(* Logix 5000 project; controller LeakTestAuto vendor 1 type 14 code 226 rev 37.11; software revision 37.01; part 14 of 14 *)
(* tags used below, declared in another part *)
   OP220 : udt_Mode;
   OP220_EStop_OK : BOOL;
   OP220_EStopTest_DCS : DCI_STOP;
   OP220_Power : BOOL;
   SI_OP220_N1_LASER_AREA_NC12 : ALIAS FOR Local:1:I.Pt00.Data;
   SI_OP220_N1_LASER_GUARD_NC12 : ALIAS FOR Local:1:I.Pt01.Data;
   SO_OP220_N2_SSR_1 : ALIAS FOR Local:2:O.Pt00.Data;
   SO_OP220_N2_SSR_2 : ALIAS FOR Local:2:O.Pt01.Data;
(* MainProgram, continued *)

ROUTINE zzUnused   (* ladder *)
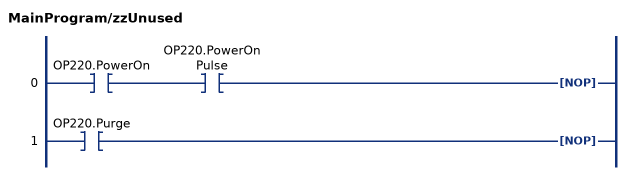
   0: XIC(OP220.PowerOn)XIC(OP220.PowerOnPulse)NOP();
   1: XIC(OP220.Purge)NOP();
END_ROUTINE
END_PROGRAM

PROGRAM SafetyProgram   (* main routine MainRoutine, safety *)
VAR
   TON_EStopFaultReset : TIMER := (PRE := 1000);
END_VAR

ROUTINE MainRoutine   (* ladder *)
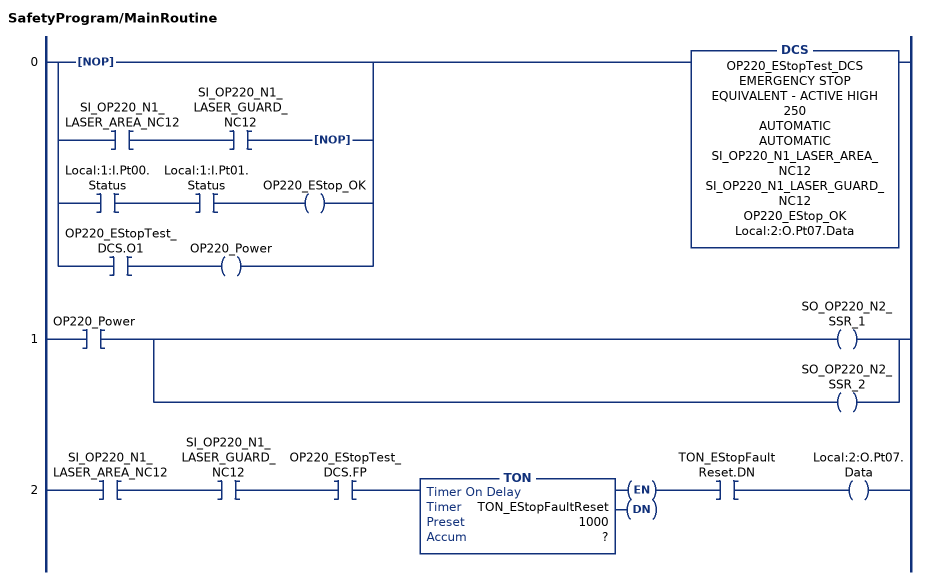
   0: [NOP() ,XIC(SI_OP220_N1_LASER_AREA_NC12) XIC(SI_OP220_N1_LASER_GUARD_NC12) NOP() ,XIC(Local:1:I.Pt00.Status) XIC(Local:1:I.Pt01.Status) OTE(OP220_EStop_OK) ,XIC(OP220_EStopTest_DCS.O1) OTE(OP220_Power) ]DCS(OP220_EStopTest_DCS,EMERGENCY STOP,EQUIVALENT - ACTIVE HIGH,250,AUTOMATIC,AUTOMATIC,SI_OP220_N1_LASER_AREA_NC12,SI_OP220_N1_LASER_GUARD_NC12,OP220_EStop_OK,Local:2:O.Pt07.Data);
   1: XIC(OP220_Power)[OTE(SO_OP220_N2_SSR_1) ,OTE(SO_OP220_N2_SSR_2) ];
   2: XIC(SI_OP220_N1_LASER_AREA_NC12)XIC(SI_OP220_N1_LASER_GUARD_NC12)XIC(OP220_EStopTest_DCS.FP)TON(TON_EStopFaultReset,?,?)XIC(TON_EStopFaultReset.DN)OTE(Local:2:O.Pt07.Data);
END_ROUTINE
END_PROGRAM
